FUNCTION_BLOCK TestModule_1
VAR_INPUT
	fbNextStationReleaseClient : ReleaseClient;
END_VAR
VAR_OUTPUT
END_VAR
VAR
END_VAR

fbNextStationReleaseClient();

END_FUNCTION_BLOCK

(* stored: Version 1.1.0.1, ProductVersion 3.1.4024.2
   POU TestModule_1: Id {31b6fd3e-e590-4345-a850-c1bd78899edc}, SpecialFunc None *)
